PROGRAM DataStorage
VAR
	fbSceneMaster	:FB_IoT_SceneMaster;
	fbTON			:TON;
	fbSceneLight	:FB_IoT_Switch(P_IoT_Com.fbIoT_ComClient,0);
	
	bWrite			:BOOL;
	bManuell		:BOOL;
END_VAR

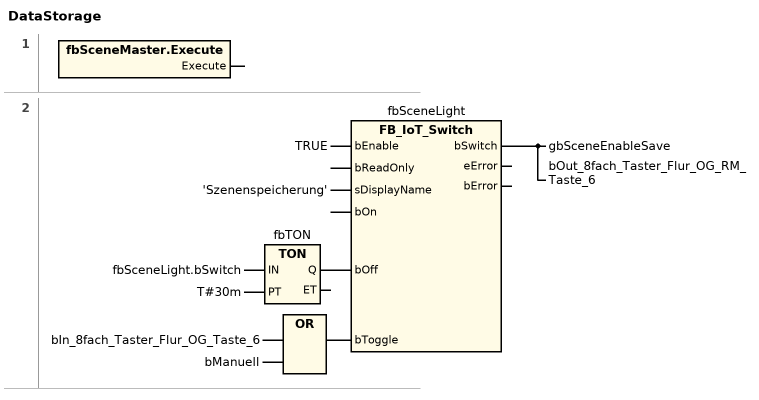
// NETWORK 1
fbSceneMaster.Execute();

// NETWORK 2
fbTON(IN := fbSceneLight.bSwitch, PT := T#30m); // TON
fbSceneLight(
    bEnable := TRUE,
    sDisplayName := 'Szenenspeicherung',
    bOff := fbTON.Q,
    bToggle := bIn_8fach_Taster_Flur_OG_Taste_6 OR bManuell); // FB_IoT_Switch
gbSceneEnableSave := fbSceneLight.bSwitch;
bOut_8fach_Taster_Flur_OG_RM_Taste_6 := fbSceneLight.bSwitch;

END_PROGRAM

(* stored: Version 1.1.0.1, ProductVersion 3.1.4024.11
   POU DataStorage: Id {40978492-2a84-4382-a701-4c1fc7c2dd4b}, SpecialFunc None *)
